TYPE ST_DALIBridgeNotification :
STRUCT
	valid 				: BOOL;
	sequence 			: ULINT;
	nInputEvents		: BYTE;
	inputEvents 		: ARRAY [0..GVL_DALIBridge.maxInputEventsPerNotification-1] OF ST_DALIBridgeInputEvent;
END_STRUCT
END_TYPE

(* stored: Version 1.1.0.1, ProductVersion 3.1.4024.11
   DUT ST_DALIBridgeNotification: Id {36c6ab18-21ed-49d0-9a4f-1fc292e884e7} *)
